INTERFACE itfFault

METHOD mResetFault : BOOL
VAR_INPUT
END_VAR
END_METHOD

METHOD mSetFault : BOOL
VAR_INPUT
END_VAR
END_METHOD

PROPERTY pFault : Bool
GET
END_GET
SET
END_SET
END_PROPERTY

PROPERTY pFaultStatus : Bool
GET
END_GET
SET
END_SET
END_PROPERTY

PROPERTY pResetButton : BOOL
GET
END_GET
SET
END_SET
END_PROPERTY

END_INTERFACE

(* stored: Version 1.1.0.1, ProductVersion 3.1.4024.12
   Itf itfFault: Id {4e737285-bd16-49a6-b68d-92a36c679a54}
   Method mResetFault: Id {da1066ea-dba9-4660-9d3b-4e357ea0a7cc}
   Method mSetFault: Id {6c7a6526-5a04-4c50-8a84-8b2f3581f2c0}
   Property pFault: Id {62823e24-0ca6-4da2-8ba6-4a5fee85736a}
   Get Get: Id {d1688689-02ad-4771-9be3-6b173b58f6ee}
   Set Set: Id {37142f89-d0da-44ec-a88d-6c793aa89fc5}
   Property pFaultStatus: Id {bd8cce7c-95d4-4838-9a36-ebe8f3175a34}
   Get Get: Id {87dc6f5c-65bf-42af-b9cf-1338e2ca41a9}
   Set Set: Id {b051b66d-27e2-4de2-b0d8-b0ef314d18b1}
   Property pResetButton: Id {0b1a16dc-8a84-4b4c-92b8-74453f94b1f8}
   Get Get: Id {cc0383d6-0e5b-4441-b42d-4d4d5cb01b14}
   Set Set: Id {d04c1f4f-4e0c-46bc-8518-c7e851718f38} *)
